FUNCTION_BLOCK FB_MultiMotorController
VAR_INPUT
	bExecute : BOOL; // Used to execute command. If error occurs excecute must go false and true again to execute command again. 
	aMotorRef :ARRAY[1..4] OF POINTER TO FB_teknicMotorEC; // Array of addresses of up to four motors to control. *Fill array in order of index **Must fill entire array. Unused spots - enter 0.
	eMethod : E_teknicMotorMethods; // Method to call for control of specified motors
END_VAR
VAR_OUTPUT
	aDone 			: ARRAY[1..4] OF BOOL;
	aBusy			: ARRAY[1..4] OF BOOL;
	aError 			: ARRAY[1..4] OF BOOL;
	aErrorID 		: ARRAY[1..4] OF UDINT;
	sControllerMsg 	: STRING; // String used to display messages from the controller FB.
END_VAR
VAR
	fbExecute 		: R_TRIG;
	bDone: INT;
END_VAR

(* Example call- FB_multiMotorController(bExecute := TRUE, aMotorRef := [ADR(FB_teknicMotor1),ADR(FB_teknicMotor2),0,0],sMethod := moveToJog); *)
fbExecute(CLK := bExecute);
IF NOT bExecute THEN
(* reset at falling edge of Execute *)
	aDone[1.4]				:= FALSE;
	aError[1.4] 			:= FALSE;
	aErrorID[1.4] 			:= 0;
END_IF
		
CASE eMethod OF 
	brakeOff://
		IF aMotorRef[1] <> 0 THEN
			aMotorRef[1]^.brakeOff();
		END_IF
		IF aMotorRef[2] <> 0 THEN
			aMotorRef[2]^.brakeOff();
		END_IF
		IF aMotorRef[3] <> 0 THEN
			aMotorRef[3]^.brakeOff();
		END_IF
		IF aMotorRef[4] <> 0 THEN
			aMotorRef[4]^.brakeOff();
		END_IF
		
	brakeOn://
		IF aMotorRef[1] <> 0 THEN
			aMotorRef[1]^.brakeOn();
		END_IF
		IF aMotorRef[2] <> 0 THEN
			aMotorRef[2]^.brakeOn();
		END_IF
		IF aMotorRef[3] <> 0 THEN
			aMotorRef[3]^.brakeOn();
		END_IF
		IF aMotorRef[4] <> 0 THEN
			aMotorRef[4]^.brakeOn();
		END_IF
		
	checkOutputs://
	coupleToAxis://
	decoupleAxis://
	disable://
	enable://
	estop://
	homeToSensor://
	homeToTorque://
	motorInit://
	moveTo://
	moveToJog://
	moveToSensor://
	moveToTorque://
	readMotorParameter://
		sControllerMsg := LREAL_TO_STRING(aMotorRef[1]^.readValue);
	removeStop://
	motorReset://
	resetMotorCommands://
	setError://
	stop://
	writeMotorParameter://
END_CASE

END_FUNCTION_BLOCK

(* stored: Version 1.1.0.1, ProductVersion 3.1.4024.15
   POU FB_MultiMotorController: Id {768fffa5-dcc7-4ac1-8696-c781292a10d5}, SpecialFunc None *)
